Universal Robots PolyScope program: Hospital_small_top.urp

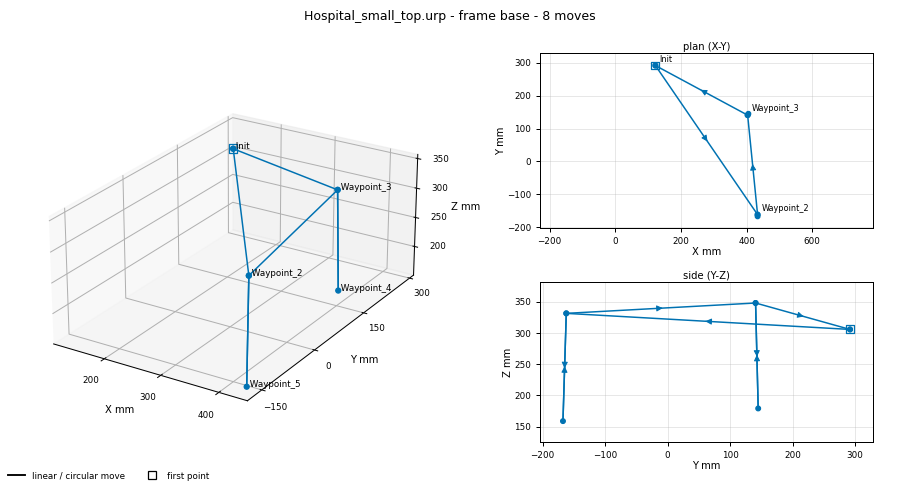
[picture p0: tool path of Hospital_small_top.urp in frame base, 8 of 8 moves have a stored position in this frame; points joined in program order, loops and branches not executed]
Program Hospital_small_top (installation=default directory=/programs/Mursal createdIn=5.11.11.1010533 lastSavedIn=5.11.11.1010533 robotSerialNumber=20205300864)
Calibrated DH parameters: a=[-0.000166, -0.243494, -0.153108, 0.000057, -0.000123, 0]; d=[0.151897, -1.34267, 53.988124, -52.514559, 0.085283, 0.092193]; alpha=[1.572472, -0.003756, 0.002824, 1.570807, -1.572621, 0]; deltaTheta=[0, 0.020704, 7.033215, -0.770746, 0.000004, 0]
Robot Program (runOnlyOnce=true)
  MoveL speed 250 mm/s, acceleration 1200 mm/s^2 (useActiveTCP=true) feature=Base
    Waypoint Init: TCP in base x=122.108 y=292.111 z=305.718 mm, rx=1.1348 ry=-2.9295 rz=0.0002 rad; joints [91.643, -87.586, -91.768, -90.547, 90.031, 859.395] deg
    Waypoint Waypoint_2: TCP in base x=433.452 y=-162.188 z=331.45 mm, rx=-2.2029 ry=-2.2398 rz=0 rad; joints [-4.055, -133.561, -19.862, -116.474, 89.813, 894.999] deg
    Waypoint Waypoint_5: TCP in base x=433.486 y=-167.49 z=158.907 mm, rx=2.2028 ry=2.2399 rz=0 rad; joints [-4.851, -132.152, -70.26, -67.482, 89.91, 894.294] deg
    URCap Gripper (Robotiq_Grippers, Robotiq Inc.) dataModel(position=75.63725490196077, force=3.0, speed=0.0, positionInDouble=75.63725490196077, forceInDouble=3.0, speedInDouble=0.0, slaveIds=[9], blocking=true, robotCompliant=false)
    Waypoint Waypoint_2: TCP in base x=433.452 y=-162.188 z=331.45 mm, rx=-2.2029 ry=-2.2398 rz=0 rad; joints [-4.055, -133.561, -19.862, -116.474, 89.813, 894.999] deg
    Waypoint Waypoint_3: TCP in base x=403.167 y=140.884 z=348.03 mm, rx=-0.0436 ry=3.1412 rz=0.0001 rad; joints [37.108, -120.238, -38.323, -111.33, 89.866, 845.559] deg
    Waypoint Waypoint_4: TCP in base x=405.374 y=145.079 z=179.205 mm, rx=-0.0268 ry=3.1414 rz=-0.0001 rad; joints [37.292, -122.238, -81.696, -65.96, 89.941, 846.445] deg
    URCap Gripper (Robotiq_Grippers, Robotiq Inc.) dataModel(position=0.0, force=1.0, speed=0.0, positionInDouble=0.0, forceInDouble=1.0, speedInDouble=0.0, slaveIds=[9], blocking=true, robotCompliant=false)
    Waypoint Waypoint_3: TCP in base x=403.167 y=140.884 z=348.03 mm, rx=-0.0436 ry=3.1412 rz=0.0001 rad; joints [37.108, -120.238, -38.323, -111.33, 89.866, 845.559] deg
    Waypoint Init: TCP in base x=122.108 y=292.111 z=305.718 mm, rx=1.1348 ry=-2.9295 rz=0.0002 rad; joints [91.643, -87.586, -91.768, -90.547, 90.031, 859.395] deg
